FUNCTION_BLOCK FB_Greaser EXTENDS FB_Device
VAR_INPUT
	i_bManCmd		:BOOL; //Purge while ON, intended for manual use
	i_tPulse		:TIME; //Purge time
END_VAR
VAR_OUTPUT
END_VAR
VAR
	tPulseTimer		:TON;
END_VAR

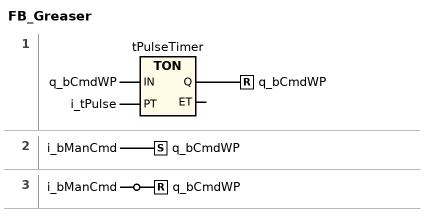
// NETWORK 1
tPulseTimer(IN := q_bCmdWP, PT := i_tPulse); // TON
q_bCmdWP R= tPulseTimer.Q;

// NETWORK 2
q_bCmdWP S= i_bManCmd;

// NETWORK 3
q_bCmdWP R= NOT i_bManCmd;

END_FUNCTION_BLOCK

(* stored: Version 1.1.0.1
   POU FB_Greaser: Id {325693c7-a385-49cc-8c68-e9ab30e8919d}, SpecialFunc None *)
